// Mitsubishi GX Works2 project: TEMPORIZADOR   PLC: Q03UDV

PROGRAM MAIN
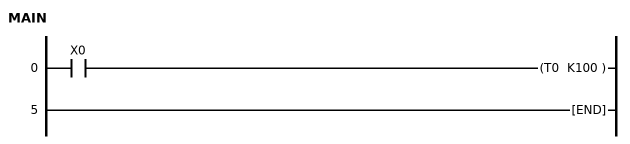
0     LD      X0
      OUT     T0 K100
5     END
END_PROGRAM
